Yaskawa INFORM job: FMTV_HOOD_TOOL_CHANGE.JBI

/JOB
//NAME FMTV_HOOD_TOOL_CHANGE
//POS
///NPOS 1,0,0,0,0,0
///TOOL 0
///POSTYPE PULSE
///PULSE
C00000=-47368,-58386,-75460,-75324,82044,-91552
//INST
///DATE 2022/03/23 12:45
///ATTR SC,RW
///GROUP1 RB1
NOP
MOVJ C00000 VJ=65.00  //TOOL CHANGE
END
